FUNCTION_BLOCK JackHAL
  (* Standard: 61499-2 *)
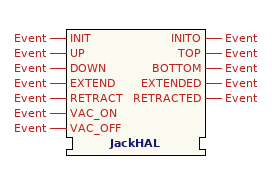
  EVENT_INPUT
    INIT;
    UP;
    DOWN;
    EXTEND;
    RETRACT;
    VAC_ON;
    VAC_OFF;
  END_EVENT
  EVENT_OUTPUT
    INITO;
    TOP;
    BOTTOM;
    EXTENDED;
    RETRACTED;
  END_EVENT
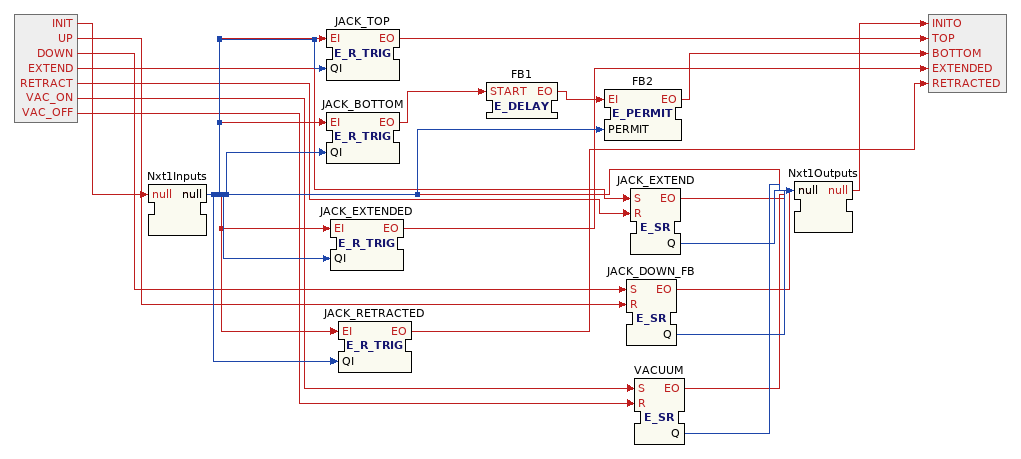
  FBS
    Nxt1Inputs : ;
    Nxt1Outputs : ;
    JACK_EXTEND : E_SR;
    JACK_DOWN_FB : E_SR;
    VACUUM : E_SR;
    JACK_EXTENDED : E_R_TRIG;
    JACK_RETRACTED : E_R_TRIG;
    JACK_TOP : E_R_TRIG;
    JACK_BOTTOM : E_R_TRIG;
    FB1 : E_DELAY;
    FB2 : E_PERMIT;
  END_FBS
  EVENT_CONNECTIONS
    INIT TO Nxt1Inputs.null;
    Nxt1Inputs.null TO Nxt1Outputs.null;
    Nxt1Outputs.null TO INITO;
    JACK_EXTEND.EO TO Nxt1Outputs.null;
    EXTEND TO JACK_EXTEND.S;
    RETRACT TO JACK_EXTEND.R;
    DOWN TO JACK_DOWN_FB.S;
    UP TO JACK_DOWN_FB.R;
    JACK_DOWN_FB.EO TO Nxt1Outputs.null;
    VACUUM.EO TO Nxt1Outputs.null;
    VAC_ON TO VACUUM.S;
    VAC_OFF TO VACUUM.R;
    JACK_EXTENDED.EO TO EXTENDED;
    JACK_RETRACTED.EO TO RETRACTED;
    Nxt1Inputs.null TO JACK_RETRACTED.EI;
    Nxt1Inputs.null TO JACK_EXTENDED.EI;
    JACK_TOP.EO TO TOP;
    JACK_BOTTOM.EO TO FB1.START;
    Nxt1Inputs.null TO JACK_TOP.EI;
    Nxt1Inputs.null TO JACK_BOTTOM.EI;
    FB1.EO TO FB2.EI;
    FB2.EO TO BOTTOM;
  END_CONNECTIONS
  DATA_CONNECTIONS
    JACK_EXTEND.Q TO Nxt1Outputs.null;
    VACUUM.Q TO Nxt1Outputs.null;
    Nxt1Inputs.null TO JACK_EXTENDED.QI;
    Nxt1Inputs.null TO JACK_RETRACTED.QI;
    Nxt1Inputs.null TO JACK_TOP.QI;
    Nxt1Inputs.null TO JACK_BOTTOM.QI;
    Nxt1Inputs.null TO FB2.PERMIT;
    JACK_DOWN_FB.Q TO Nxt1Outputs.null;
  END_CONNECTIONS
END_FUNCTION_BLOCK
